FUNCTION_BLOCK FB_ResetSequenceTestDouble IMPLEMENTS I_ResetSequence
VAR
    bIsResetted : BOOL;
END_VAR

METHOD IsReset : BOOL
IsReset := THIS^.bIsResetted;
END_METHOD

METHOD PUBLIC SetIsReset
VAR_INPUT
    bIsReset : BOOL;
END_VAR
THIS^.bIsResetted := bIsReset;
END_METHOD

END_FUNCTION_BLOCK

(* stored: Version 1.1.0.1
   POU FB_ResetSequenceTestDouble: Id {58d809bf-6ec0-41bb-8ea6-69586d794719}, SpecialFunc None
   Method IsReset: Id {d24bf294-3201-40ef-be1e-9234974ae659}
   Method SetIsReset: Id {02c6dcbb-7cb3-4c7b-9cc2-3e312fb966d9} *)
